(* IEC 61131-3 sources: AXOpen/src/components.abb.robotics/ctrl/src/AxoOmnicore/TypesStructuresAndEnums, 1 file *)

(* ---- AxoOmnicore_v_1_x_x_HWIDs.st ---- *)
NAMESPACE AXOpen.Components.Abb.Robotics
{S7.extern=ReadWrite}
CLASS AxoOmnicore_v_1_x_x_HWIDs
  VAR PUBLIC
     {#ix-set:AttributeName = "<#Hardware ID of the device#>"}
     HW_Device              :  UINT;
     {#ix-set:AttributeName = "<#Hardware ID of the 'DI_64_bytes' submodule#>"}
     HwID_DI_64_bytes       :   UINT;
     {#ix-set:AttributeName = "<#Hardware ID of the 'DO_64_bytes' submodule#>"}
     HwID_DO_64_bytes          :   UINT;
  END_VAR
END_CLASS
END_NAMESPACE
